// Mitsubishi GX Works2 project: FrekvensMLD   PLC: FX1S

// global labels: Global1
VAR_GLOBAL
  Sens_1 AT X002 : BOOL;
  Sens_2 AT X003 : BOOL;
  Sens_3 AT X004 : BOOL;
  Sens_4 AT X005 : BOOL;
  Start AT X000 : BOOL;
  Reset AT X001 : BOOL;
  Stage_1 AT M0 : BOOL;
  Stage_2 AT M1 : BOOL;
  Stage_3 AT M2 : BOOL;
  Stage_4 AT M3 : BOOL;
  Stage_5 AT M4 : BOOL;
  Stage_6 AT M5 : BOOL;
  Stage_7 AT M6 : BOOL;
  Forward AT Y000 : BOOL;
  Back AT Y001 : BOOL;
  F1 AT Y003 : BOOL;  (* Hastighet 1 *)
  F2 AT Y002 : BOOL;  (* Hastighet 2 *)
  F3 AT Y004 : BOOL;  (* Hastighet 3 *)
END_VAR

// task Task_01 (event TRUE, interval 0, priority 31): Sequence, Activation

PROGRAM Sequence
VAR
  Run : BOOL;
  Seq_Ct : CTU;
  Timer_In : TON;
END_VAR
(* structured ladder/FBD written out as ST: instructions are called as NAME(EN, inputs, outputs); _pN, _eN, _tN stand for wires *)
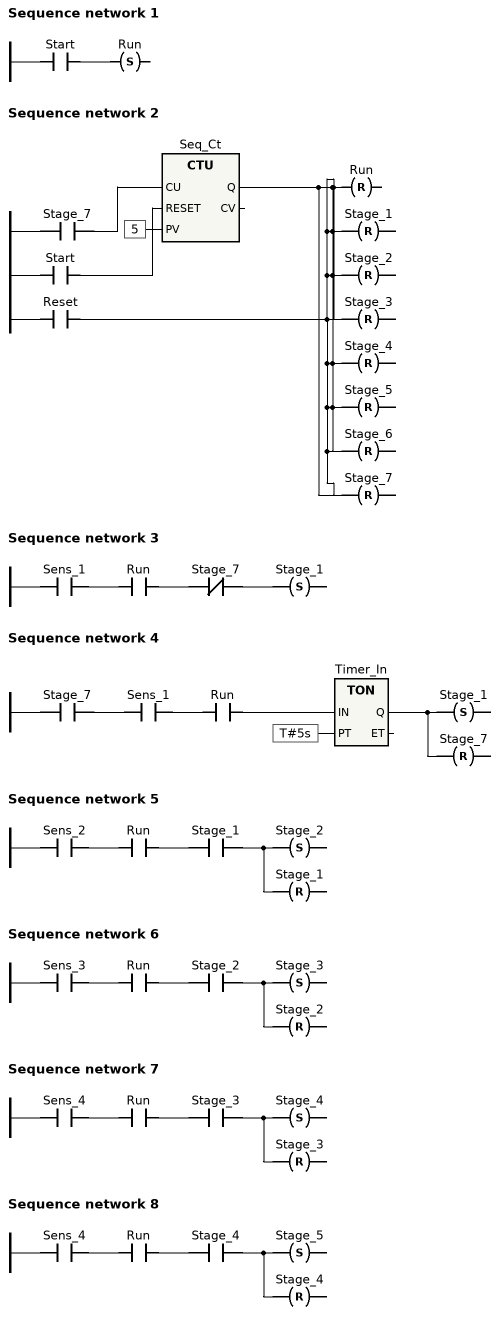
(* network 1 *)
SET(Start, Run);
(* network 2 *)
Seq_Ct(CU := Stage_7, RESET := Start, PV := 5);
_p1 := Seq_Ct.Q OR Reset;
RST(_p1, Run);
RST(_p1, Stage_1);
RST(_p1, Stage_2);
RST(_p1, Stage_3);
RST(_p1, Stage_4);
RST(_p1, Stage_5);
RST(_p1, Stage_6);
RST(_p1, Stage_7);
(* network 3 *)
SET(Sens_1 AND Run AND NOT Stage_7, Stage_1);
(* network 4 *)
Timer_In(IN := Stage_7 AND Sens_1 AND Run, PT := T#5s);
SET(Timer_In.Q, Stage_1);
RST(Timer_In.Q, Stage_7);
(* network 5 *)
_p1 := Sens_2 AND Run AND Stage_1;
SET(_p1, Stage_2);
RST(_p1, Stage_1);
(* network 6 *)
_p1 := Sens_3 AND Run AND Stage_2;
SET(_p1, Stage_3);
RST(_p1, Stage_2);
(* network 7 *)
_p1 := Sens_4 AND Run AND Stage_3;
SET(_p1, Stage_4);
RST(_p1, Stage_3);
(* network 8 *)
_p1 := Sens_4 AND Run AND Stage_4;
SET(_p1, Stage_5);
RST(_p1, Stage_4);
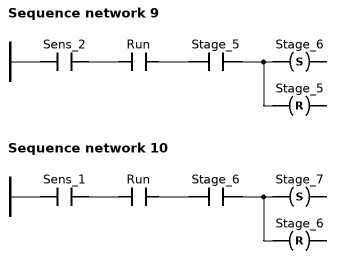
(* network 9 *)
_p1 := Sens_2 AND Run AND Stage_5;
SET(_p1, Stage_6);
RST(_p1, Stage_5);
(* network 10 *)
_p1 := Sens_1 AND Run AND Stage_6;
SET(_p1, Stage_7);
RST(_p1, Stage_6);
END_PROGRAM

PROGRAM Activation
VAR
  Timer_Out : TON;
END_VAR
(* structured ladder/FBD written out as ST: instructions are called as NAME(EN, inputs, outputs); _pN, _eN, _tN stand for wires *)
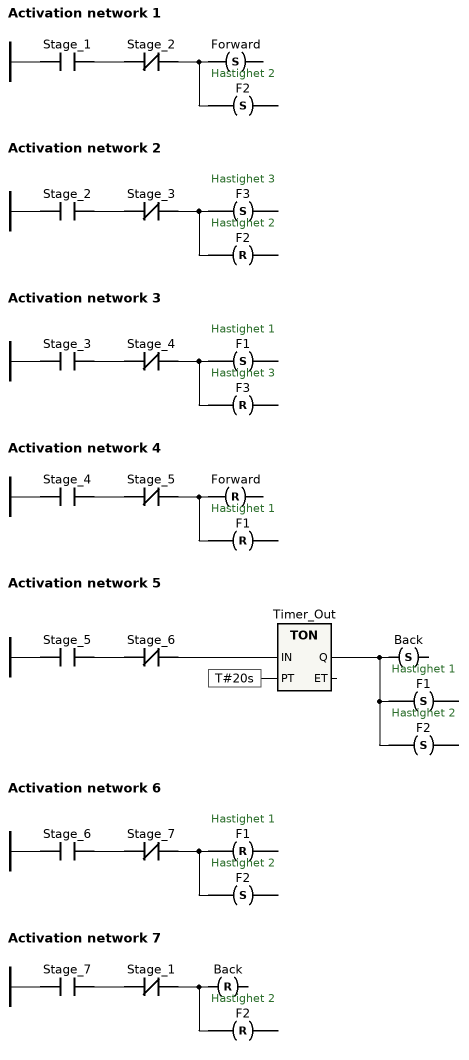
(* network 1 *)
_p1 := Stage_1 AND NOT Stage_2;
SET(_p1, Forward);
SET(_p1, F2);
(* network 2 *)
_p1 := Stage_2 AND NOT Stage_3;
SET(_p1, F3);
RST(_p1, F2);
(* network 3 *)
_p1 := Stage_3 AND NOT Stage_4;
SET(_p1, F1);
RST(_p1, F3);
(* network 4 *)
_p1 := Stage_4 AND NOT Stage_5;
RST(_p1, Forward);
RST(_p1, F1);
(* network 5 *)
Timer_Out(IN := Stage_5 AND NOT Stage_6, PT := T#20s);
SET(Timer_Out.Q, Back);
SET(Timer_Out.Q, F1);
SET(Timer_Out.Q, F2);
(* network 6 *)
_p1 := Stage_6 AND NOT Stage_7;
RST(_p1, F1);
SET(_p1, F2);
(* network 7 *)
_p1 := Stage_7 AND NOT Stage_1;
RST(_p1, Back);
RST(_p1, F2);
END_PROGRAM
